PROGRAM Dtank_Length
VAR
    setPos : MC_SetPosition;
    nominalPosition : LREAL := 2289.15;
END_VAR

GVL.astAxes[AXIS_DTANK_LENGTH].stInputs.bLimitBwd := TRUE;
GVL.astAxes[AXIS_DTANK_LENGTH].stInputs.bLimitFwd := TRUE;
GVL.astAxes[AXIS_DTANK_LENGTH].stControl.bEnable := TRUE;




IF _TaskInfo[fbGetCurTaskIndex.index].FirstCycle THEN
    //Initial default values:
    setPos.Execute:= TRUE;
END_IF


setPos.Position := nominalPosition;

setPos(Axis:= astAxes[AXIS_DTANK_LENGTH].Axis);
setPos.Execute:= FALSE;

END_PROGRAM

(* stored: Version 1.1.0.1, ProductVersion 3.1.4024.11
   POU Dtank_Length: Id {89d9baec-ea80-4314-a7ab-842a813f72f1}, SpecialFunc None *)
